FUNCTION_BLOCK FB_AUT_125 EXTENDS FB_AUT_ABSTRACT
(****************************************************************************)
(*	POU_AUT_zxx			Bausteinaufrufe Station	zxx							*)
(*	Status				ungetestet											*)
(*  Version:			1.0													*)
(*	Beschrieb:																*)
(*																			*)
(*	Abläufe:			FB_ABLzxxA		Hauptablauf							*)
(*																			*)
(*																			*)
(* 	25.09.2019/Dj															*)
(****************************************************************************)
(*	dd.mm.yyyy   KZ    x.y			Beschrieb								*)
(****************************************************************************)
VAR_INPUT
    (* spezifische Eingänge *)

END_VAR
VAR_OUTPUT
    (* spezifische Ausgänge *)

END_VAR
VAR
    (* Bausteine *)
    fb_Pnp : FB_ABL_125_Pnp;
    fb_Feeder : FB_ABL_125_Feeder;
	
END_VAR

(*******************************************************************)
(* Timer *)
(*******************************************************************)

(*******************************************************************)
(* Flanken / Merker *)
(*******************************************************************)
//MANU CYCLE
IF (enIN_State = StateMANU) AND xIN_ManuCycle THEN
    xManuCycle := TRUE;
END_IF;

IF (enIN_State <> StateMANU) OR xOUT_Done THEN
    xManuCycle := FALSE;
END_IF

//NEXT STEP
xNextStep := (enIN_State > StateSTEP) OR
             ((enIN_State = StateSTEP) AND xIN_Step) OR
             ((enIN_State = StateMANU) AND xManuCycle);

//RESET
xReset := ((enIN_State < StateREADY) AND (enIN_State <> StateINIT)) OR
          ((enIN_State = StateMANU) AND NOT xManuCycle);

(*******************************************************************)
(* Bausteinaufrufe Abläufe *)
(*******************************************************************)

fb_Pnp(xIN_Reset          := HMI.btArMain[7].on,
       xIN_Init           := xIN_Init,
       xIN_Quit           := xIN_Quit,
       xIN_Start          := enIN_State = enState.StateAUTO, //AND _FB_ABL_100A.xOUT_Done AND _FB_ABL_100A.xOUT_Ready,
       xIN_Sperre         := NOT xIN_On,
       xIN_NextStep       := xNextStep,
       xIN_AlarmAktiv     := xIN_AlarmAktiv,
       xIN_DryCycle       := xIN_DryCycle,
       xIN_RestartCYCL    := enIN_State = enState.StateAUTO, // only restart when the mover has move out
       enIN_State         := enIN_State,
       tIN_Timeout        := tIN_Timeout,
       pxFG_Freigabe      := ADR(xDummy),
       Mover              := THIS^.Mover,
       xIN_PceReadyToPick := fb_Feeder.xOUT_Done);

fb_Feeder(xIN_Reset       := HMI.btArMain[7].on,
          xIN_Init        := xIN_Init,
          xIN_Quit        := xIN_Quit,
          xIN_Start       := enIN_State = enState.StateAUTO, //AND _FB_ABL_100A.xOUT_Done AND _FB_ABL_100A.xOUT_Ready, 
          xIN_Sperre      := NOT xIN_On,
          xIN_NextStep    := xNextStep,
          xIN_AlarmAktiv  := xIN_AlarmAktiv,
          xIN_DryCycle    := xIN_DryCycle,
          xIN_RestartCYCL := enIN_State = enState.StateAUTO, // only restart when the mover has move out
          enIN_State      := enIN_State,
          tIN_Timeout     := tIN_Timeout,
          pxFG_Freigabe   := ADR(xDummy),
          xIN_PickPiece   := fb_Pnp.xOUT_PickPiece);

(*******************************************************************)
(* Mover reset flags *)
(*******************************************************************)

(*******************************************************************)
(* OUTPUT *)
(*******************************************************************)
xOUT_InitDone := fb_Pnp.xOUT_InitDone AND fb_Feeder.xOUT_InitDone;
xOUT_Ready    := xOUT_InitDone;
xOUT_Done     := fb_Pnp.xOUT_Done;
xOUT_ErrFlag  := fb_Pnp.xOUT_ErrFlag;
xOUT_Wait     := fb_Pnp.xOUT_Wait;
xOUT_AlarmST  := xOUT_ErrFlag;

(*******************************************************************)
(* Bausteinaufruf Error Station *)
(*******************************************************************)
// POU_ERR_VORLAGE(xIN_QUIT:=xIN_Quit , pstrArIN_ALARM:=ADR(HMI.strArALARM[1]));

METHOD GiveMover : IProcessSampleMover
VAR_INPUT
	mover : REFERENCE TO FB_Mover;
END_VAR
IF __ISVALIDREF(mover) THEN
    THIS^.Mover                       REF= mover;
END_IF
END_METHOD

(* % of completion of the process *)
PROPERTY iCompletionPC : INT
GET
iCompletionPC := THIS^.fb_Pnp.iOUT_ProcessCompletion;
END_GET
END_PROPERTY

PROPERTY ProcessExecution : ProcessExecution_e
GET
ProcessExecution := THIS^._ProcessExecution;
END_GET
SET
THIS^._ProcessExecution := ProcessExecution;
END_SET
END_PROPERTY

METHOD TakeMover : IProcessSampleMover
VAR_INPUT
END_VAR
THIS^.Mover REF= 0;
END_METHOD

PROPERTY xBusy : BOOL
GET
xBusy := THIS^.fb_Pnp.xOUT_Busy;
END_GET
SET
END_SET
END_PROPERTY

PROPERTY xDone : BOOL
GET
xDone := THIS^.fb_Pnp.xOUT_Ready OR THIS^.fb_Pnp.xOUT_Done;
END_GET
END_PROPERTY

PROPERTY xMoverPathFree : BOOL
GET
xMoverPathFree := THIS^.fb_Pnp.xOUT_MoverFree OR THIS^.fb_Pnp.xOUT_Ready OR THIS^.fb_Pnp.xOUT_Done;
END_GET
END_PROPERTY

PROPERTY xMoverShouldLeave : BOOL
GET
xMoverShouldLeave := THIS^.fb_Pnp.iOUT_Step = ST125_Pnp_e.SYNC_MOVER_LEAVE;
END_GET
END_PROPERTY

END_FUNCTION_BLOCK

(* stored: Version 1.1.0.1, ProductVersion 3.1.4024.6
   POU FB_AUT_125: Id {983e6e7a-a005-4f39-ac41-ff8b5e2a2f31}, SpecialFunc None
   Method GiveMover: Id {42a78642-302d-4ed6-89d5-c3491d94d870}
   Property iCompletionPC: Id {b75bbe01-24aa-4e4b-b51b-e0c348230a53}
   Get Get: Id {cbdf50a6-757a-464e-a6b6-2c796c025af5}
   Property ProcessExecution: Id {b4cce3de-8f2c-468e-b36e-fe342b32d58d}
   Get Get: Id {3a1dcd01-7749-48bc-b084-84585759f5c2}
   Set Set: Id {e3df0f3e-a786-416d-97db-1a9cbe3b8e6c}
   Method TakeMover: Id {e9b56a9b-1da7-4fef-b8b9-4f9c3ad58499}
   Property xBusy: Id {f6ad6f68-d20d-4fae-8dbe-ff523afc20f2}
   Get Get: Id {672e506d-5782-4369-ab59-bd2dfbe69ab5}
   Set Set: Id {93ff59b2-de16-46da-85b3-89d7e1d45976}
   Property xDone: Id {da9a93d0-1c56-456b-9380-02f239d53e98}
   Get Get: Id {27c3ca5e-6bdd-4e12-983d-db8716759355}
   Property xMoverPathFree: Id {74eb02b6-b0e5-46e8-937f-4096b526318f}
   Get Get: Id {f4e9ec5c-3c33-4c39-93bf-8191bf1db9fc}
   Property xMoverShouldLeave: Id {ffbf91fc-ffe7-4388-bb2f-ca66cf2673c0}
   Get Get: Id {60ee839c-8ead-4d6d-a398-eb399edf2d00} *)
